ABB RAPID module: 005_home_corner_square_v2.mod

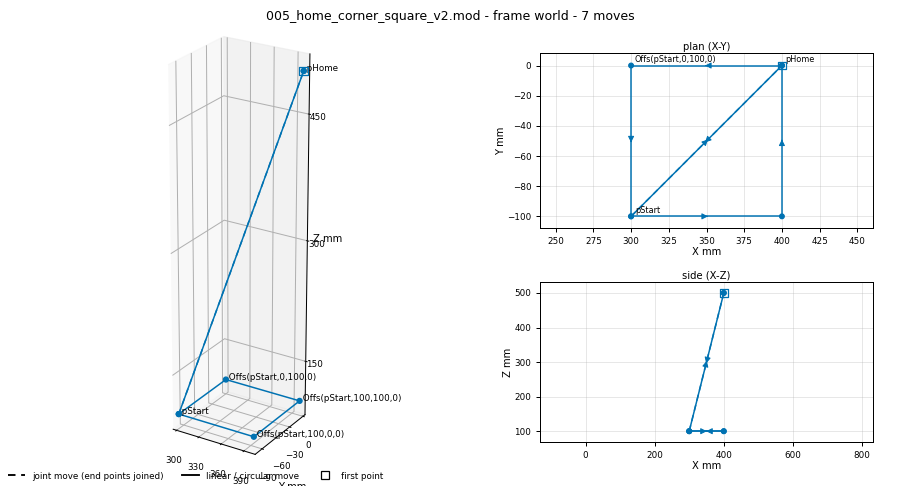
[picture p0: tool path of 005_home_corner_square_v2.mod in frame world, 7 of 7 moves have a stored position in this frame; points joined in program order, loops and branches not executed]
MODULE Ex005_HomeCornerSquare
! Exercise 5 - Home corner square
! Move to a safe home position then draw a 100 x 100 square using RelTool offsets

  PERS robtarget pHome  := [[400, 0, 500], [1,0,0,0], [0,0,0,0], [9E9,9E9,9E9,9E9,9E9,9E9]];
  PERS robtarget pStart := [[300, -100, 100], [1,0,0,0], [0,0,0,0], [9E9,9E9,9E9,9E9,9E9,9E9]];

  PROC Ex005_Run()
      ! 1. Safe approach to home position (joint motion, fast)
      MoveJ pHome, v500, z50, tool0;        ! tool0 = default tool

      ! 2. Move linearly to the first corner of the square (precise stop)
      MoveL pStart, v100, fine, tool0;

      ! 3. Trace the square from pStart (X, Y, Z)
      MoveL Offs(pStart, 100, 0, 0), v100, z1, tool0;    ! Move along X (right, corner 2)
      MoveL Offs(pStart, 100, 100, 0), v100, z1, tool0;  ! Move along Y (forward, corner 3)
      MoveL Offs(pStart, 0, 100, 0), v100, z1, tool0;    ! Move along X (Left, corner 4)
      MoveL pStart, v100, fine, tool0;    ! Move along Y (Back to pStart, corner 1)

      ! 4. Return to safe home position
      MoveJ pHome, v500, z50, tool0;

  ENDPROC

ENDMODULE
